FUNCTION_BLOCK FB_LowVoltageMainDistribution
VAR_INPUT
END_VAR
VAR_OUTPUT
END_VAR
VAR
	EM_Offices : FB_ElectricityMeter_ABBA44113100;
	EM_ProductionHall_HVAC : FB_ElectricityMeter_ABBA44113100;
	EM_ProductionHall_Lighting : FB_ElectricityMeter_ABBA44113100;
	EM_TotalBuilding : FB_ElectricityMeter_ABBA44213100;
END_VAR

EM_Offices(aElectricityMeterTelegramm := Telegramm_SZ_Buerotrakt);
EM_ProductionHall_HVAC(aElectricityMeterTelegramm := Telegramm_SZ_Halle_TGA);
EM_ProductionHall_Lighting(aElectricityMeterTelegramm := Telegramm_SZ_Halle_Licht);
EM_TotalBuilding(aElectricityMeterTelegramm := Telegramm_SZ_Gebaeude);

END_FUNCTION_BLOCK

(* stored: Version 1.1.0.1, ProductVersion 3.1.4024.10
   POU FB_LowVoltageMainDistribution: Id {65b26091-d75a-4596-946d-a290447522cb}, SpecialFunc None *)
